{attribute addProperty BoxType "EJ6910-0000-0018"}
{attribute addProperty Id "FSLOGIC_InputsAT %I*FSLOGIC_Inputs_8BA5C9331620FSLOGIC_OutputsAT %Q*EMPTY_STRUCTURE000WcStateAT %I*WcState_F855686C1620InfoDataAT %I*InfoData_BC63D37F80100"}
{attribute addProperty CRC "2883950380"}
{attribute addProperty SizeInBites "112"}
{attribute addProperty SizeInBytes "14"}
TYPE EJ6910_13AA9334 :
STRUCT
	{attribute addProperty Name "FSLOGIC_Inputs"}
	FSLOGIC_Inputs : FSLOGIC_Inputs_8BA5C933;
	{attribute addProperty Name "FSLOGIC_Outputs"}
	FSLOGIC_Outputs : EMPTY_STRUCTURE;
	{attribute addProperty Name "WcState"}
	WcState : WcState_F855686C;
	{attribute addProperty Name "InfoData"}
	InfoData : InfoData_BC63D37F;
END_STRUCT
END_TYPE

(* stored: Version 1.2.0.0, ProductVersion 3.1.4024.9
   DUT EJ6910_13AA9334: Id {51ccf109-94f3-4147-b297-9fba6d5ab18d} *)
